PROGRAM MAIN
VAR
	Check			:BOOL;
END_VAR

Anlage();

END_PROGRAM

(* stored: Version 1.1.0.1, ProductVersion 3.1.4024.12
   POU MAIN: Id {d5feccea-6762-47e0-99a4-b2697d0f6092}, SpecialFunc None *)
